(* IEC 61131-3 sources: volt/packages/volt-lsp-iec/test-corpus/bakon-nano/Device/Plc Logic/Application/Library Manager/SysDir, 15 files *)

(* ---- DIRFILETIME.dut ---- *)
TYPE DIRFILETIME :
STRUCT
	ULCREATION : UDINT;
	ULLASTACCESS : UDINT;
	ULLASTMODIFICATION : UDINT;
END_STRUCT
END_TYPE

(* ---- DIRINFO.dut ---- *)
TYPE DIRINFO :
STRUCT
	TDIRFILETIME : DirFileTime;
	ULSIZE : __XWORD;
	DIDIRECTORY : DINT;
END_STRUCT
END_TYPE

(* ---- DIRINFOFLAGS.gvl ---- *)
VAR_GLOBAL
	DF_FILE : DWORD := 16#0;
	DF_DIRECTORY : DWORD := 16#2;
END_VAR

(* ---- GVL.gvl ---- *)
VAR_GLOBAL
	SYSDIR_INVALID_HANDLE : RTS_IEC_HANDLE := RTS_INVALID_HANDLE;
END_VAR

(* ---- SYSDIRCLOSE.pou ---- *)
FUNCTION SYSDIRCLOSE : RTS_IEC_RESULT
VAR_INPUT
	HDIR : RTS_IEC_HANDLE;
END_VAR
END_FUNCTION

(* ---- SYSDIRCOPY.pou ---- *)
FUNCTION SYSDIRCOPY : RTS_IEC_RESULT
VAR_INPUT
	SZDESTDIR : REFERENCE TO STRING;
	SZSOURCEDIR : REFERENCE TO STRING;
	XRECURSIVE : BOOL;
	XOVERWRITE : BOOL;
END_VAR
END_FUNCTION

(* ---- SYSDIRCREATE.pou ---- *)
FUNCTION SYSDIRCREATE : RTS_IEC_RESULT
VAR_INPUT
	SZDIR : REFERENCE TO STRING;
END_VAR
END_FUNCTION

(* ---- SYSDIRCREATE2.pou ---- *)
FUNCTION SYSDIRCREATE2 : RTS_IEC_RESULT
VAR_INPUT
	SZDIR : REFERENCE TO STRING;
	XRECURSIVE : BOOL;
END_VAR
END_FUNCTION

(* ---- SYSDIRDELETE.pou ---- *)
FUNCTION SYSDIRDELETE : RTS_IEC_RESULT
VAR_INPUT
	SZDIR : REFERENCE TO STRING;
END_VAR
END_FUNCTION

(* ---- SYSDIRDELETE2.pou ---- *)
FUNCTION SYSDIRDELETE2 : RTS_IEC_RESULT
VAR_INPUT
	SZDIR : REFERENCE TO STRING;
	XRECURSIVE : BOOL;
	XKEEPDIR : BOOL;
END_VAR
END_FUNCTION

(* ---- SYSDIRGETCURRENT.pou ---- *)
FUNCTION SYSDIRGETCURRENT : RTS_IEC_RESULT
VAR_INPUT
	DIMAXDIRLEN : DINT;
END_VAR
VAR_IN_OUT
	SZDIR : STRING;
END_VAR
END_FUNCTION

(* ---- SYSDIROPEN.pou ---- *)
FUNCTION SYSDIROPEN : RTS_IEC_HANDLE
VAR_INPUT
	SZDIR : REFERENCE TO STRING;
	SZDIRENTRY : REFERENCE TO STRING;
	DIMAXDIRENTRY : DINT;
	PDIRINFO : POINTER TO DirInfo;
	PRESULT : POINTER TO RTS_IEC_RESULT;
END_VAR
END_FUNCTION

(* ---- SYSDIRREAD.pou ---- *)
FUNCTION SYSDIRREAD : RTS_IEC_RESULT
VAR_INPUT
	HDIR : RTS_IEC_HANDLE;
	DIMAXDIRENTRY : DINT;
	PDIRINFO : POINTER TO DirInfo;
END_VAR
VAR_IN_OUT
	SZDIRENTRY : STRING;
END_VAR
END_FUNCTION

(* ---- SYSDIRRENAME.pou ---- *)
FUNCTION SYSDIRRENAME : RTS_IEC_RESULT
VAR_INPUT
	SZOLDDIRNAME : REFERENCE TO STRING;
	SZNEWDIRNAME : REFERENCE TO STRING;
END_VAR
END_FUNCTION

(* ---- SYSDIRSETCURRENT.pou ---- *)
FUNCTION SYSDIRSETCURRENT : RTS_IEC_RESULT
VAR_INPUT
	SZDIR : REFERENCE TO STRING;
END_VAR
END_FUNCTION
